SUBAPPLICATION AX_2_2 (* AX_OR and AX_SPLIT for a 2-to-2 Connection *)
  (* Standard: 61499-2 *)
  (* Version 1.0, 2026-05-29, franz, Meisterschulen am Ostbahnhof *)
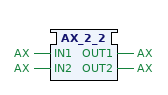
  SOCKETS
    IN1 : adapter::types::unidirectional::AX;
    IN2 : adapter::types::unidirectional::AX;
  END_SOCKETS
  PLUGS
    OUT1 : adapter::types::unidirectional::AX;
    OUT2 : adapter::types::unidirectional::AX;
  END_PLUGS
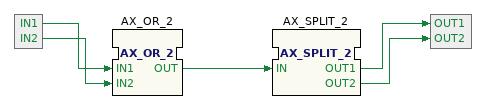
  FBS
    AX_SPLIT_2 : adapter::events::unidirectional::AX_SPLIT_2;
    AX_OR_2 : adapter::booleanOperators::AX_OR_2;
  END_FBS
  ADAPTER_CONNECTIONS
    AX_OR_2.OUT TO AX_SPLIT_2.IN;
    AX_SPLIT_2.OUT1 TO OUT1;
    AX_SPLIT_2.OUT2 TO OUT2;
    IN1 TO AX_OR_2.IN1;
    IN2 TO AX_OR_2.IN2;
  END_CONNECTIONS
END_SUBAPPLICATION
